TYPE COMPLEX :
STRUCT
	re : REAL;
	im : REAL;
END_STRUCT
END_TYPE

(* stored: Version 1.1.0.1, ProductVersion 3.1.4024.9
   DUT COMPLEX: Id {6c3e51ae-c1ad-43ae-9fd3-1c331116ee91} *)
